// TIA Portal V16 export
// export: Created 2021-11-12T13:31:07.6036051Z, ExportSetting WithDefaults, DisplayName Totally Integrated Automation Portal, DisplayVersion V16 Update 3, DisplayName TIA Portal Version Control Interface, DisplayVersion V16 Update 2, DisplayName TIA Portal Openness, DisplayVersion V16 Update 3, DisplayName SINAMICS Startdrive Advanced, DisplayVersion V16 Update 5, DisplayName SINAMICS Startdrive G130, G150, S120, S150, SINAMICS MV, S210, DisplayVersion V16 Update 5, DisplayName SINAMICS Startdrive G110M, G120, G120C, G120D, G120P, G115D, DisplayVersion V16 Update 5, DisplayName STEP 7 Professional, DisplayVersion V16 Update 3, DisplayName STEP 7 Safety, DisplayVersion V16, DisplayName WinCC UA Professional, DisplayVersion V16 Update 3
FUNCTION_BLOCK "Sfty_IO_Module"   // FB68, F_LAD
{ S7_Optimized_Access := 'TRUE' }
VERSION : 0.1
// Safety module fault evaluation
// stored: AutoNumber true, IsIECCheckEnabled false, UDAEnableTagReadback false
   VAR
      SF_AckGlobal : ACK_GL;
   END_VAR
BEGIN

REGION Network 2: Acknowledgment for reintegration
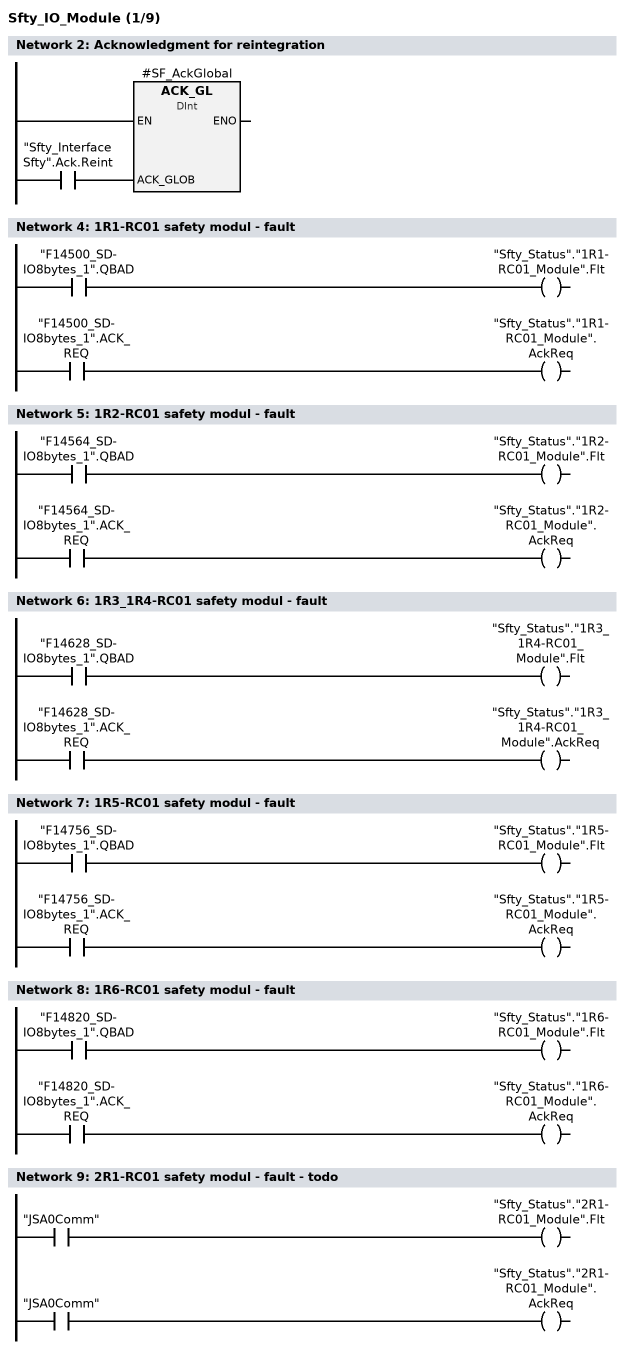
   RUNG wire#powerrail
      { S7_Templates := "codedbool_type := DInt" } #SF_AckGlobal.ACK_GL(ACK_GLOB := wire#w1)
   END_RUNG
   RUNG wire#powerrail
      Contact( "Sfty_InterfaceSfty".Ack.Reint )
   END_RUNG wire#w1
   // the same network as SCL:
   #SF_AckGlobal(ACK_GLOB := "Sfty_InterfaceSfty".Ack.Reint);   // ACK_GL
END_REGION

REGION Network 3: *************** Robot safety module fault ***************
END_REGION

REGION Network 4: 1R1-RC01 safety modul - fault
   RUNG wire#powerrail
      Contact( "F14500_SD-IO8bytes_1".QBAD )
      Coil( "Sfty_Status"."1R1-RC01_Module".Flt )
   END_RUNG
   RUNG wire#powerrail
      Contact( "F14500_SD-IO8bytes_1".ACK_REQ )
      Coil( "Sfty_Status"."1R1-RC01_Module".AckReq )
   END_RUNG
   // the same network as SCL:
   "Sfty_Status"."1R1-RC01_Module".Flt := "F14500_SD-IO8bytes_1".QBAD;
   "Sfty_Status"."1R1-RC01_Module".AckReq := "F14500_SD-IO8bytes_1".ACK_REQ;
END_REGION

REGION Network 5: 1R2-RC01 safety modul - fault
   RUNG wire#powerrail
      Contact( "F14564_SD-IO8bytes_1".QBAD )
      Coil( "Sfty_Status"."1R2-RC01_Module".Flt )
   END_RUNG
   RUNG wire#powerrail
      Contact( "F14564_SD-IO8bytes_1".ACK_REQ )
      Coil( "Sfty_Status"."1R2-RC01_Module".AckReq )
   END_RUNG
   // the same network as SCL:
   "Sfty_Status"."1R2-RC01_Module".Flt := "F14564_SD-IO8bytes_1".QBAD;
   "Sfty_Status"."1R2-RC01_Module".AckReq := "F14564_SD-IO8bytes_1".ACK_REQ;
END_REGION

REGION Network 6: 1R3_1R4-RC01 safety modul - fault
   RUNG wire#powerrail
      Contact( "F14628_SD-IO8bytes_1".QBAD )
      Coil( "Sfty_Status"."1R3_1R4-RC01_Module".Flt )
   END_RUNG
   RUNG wire#powerrail
      Contact( "F14628_SD-IO8bytes_1".ACK_REQ )
      Coil( "Sfty_Status"."1R3_1R4-RC01_Module".AckReq )
   END_RUNG
   // the same network as SCL:
   "Sfty_Status"."1R3_1R4-RC01_Module".Flt := "F14628_SD-IO8bytes_1".QBAD;
   "Sfty_Status"."1R3_1R4-RC01_Module".AckReq := "F14628_SD-IO8bytes_1".ACK_REQ;
END_REGION

REGION Network 7: 1R5-RC01 safety modul - fault
   RUNG wire#powerrail
      Contact( "F14756_SD-IO8bytes_1".QBAD )
      Coil( "Sfty_Status"."1R5-RC01_Module".Flt )
   END_RUNG
   RUNG wire#powerrail
      Contact( "F14756_SD-IO8bytes_1".ACK_REQ )
      Coil( "Sfty_Status"."1R5-RC01_Module".AckReq )
   END_RUNG
   // the same network as SCL:
   "Sfty_Status"."1R5-RC01_Module".Flt := "F14756_SD-IO8bytes_1".QBAD;
   "Sfty_Status"."1R5-RC01_Module".AckReq := "F14756_SD-IO8bytes_1".ACK_REQ;
END_REGION

REGION Network 8: 1R6-RC01 safety modul - fault
   RUNG wire#powerrail
      Contact( "F14820_SD-IO8bytes_1".QBAD )
      Coil( "Sfty_Status"."1R6-RC01_Module".Flt )
   END_RUNG
   RUNG wire#powerrail
      Contact( "F14820_SD-IO8bytes_1".ACK_REQ )
      Coil( "Sfty_Status"."1R6-RC01_Module".AckReq )
   END_RUNG
   // the same network as SCL:
   "Sfty_Status"."1R6-RC01_Module".Flt := "F14820_SD-IO8bytes_1".QBAD;
   "Sfty_Status"."1R6-RC01_Module".AckReq := "F14820_SD-IO8bytes_1".ACK_REQ;
END_REGION

REGION Network 9: 2R1-RC01 safety modul - fault - todo
   RUNG wire#powerrail
      Contact( "JSA0Comm" )
      Coil( "Sfty_Status"."2R1-RC01_Module".Flt )
   END_RUNG
   RUNG wire#powerrail
      Contact( "JSA0Comm" )
      Coil( "Sfty_Status"."2R1-RC01_Module".AckReq )
   END_RUNG
   // the same network as SCL:
   "Sfty_Status"."2R1-RC01_Module".Flt := "JSA0Comm";
   "Sfty_Status"."2R1-RC01_Module".AckReq := "JSA0Comm";
END_REGION

REGION Network 10: 2R2-RC01 safety modul - fault - todo
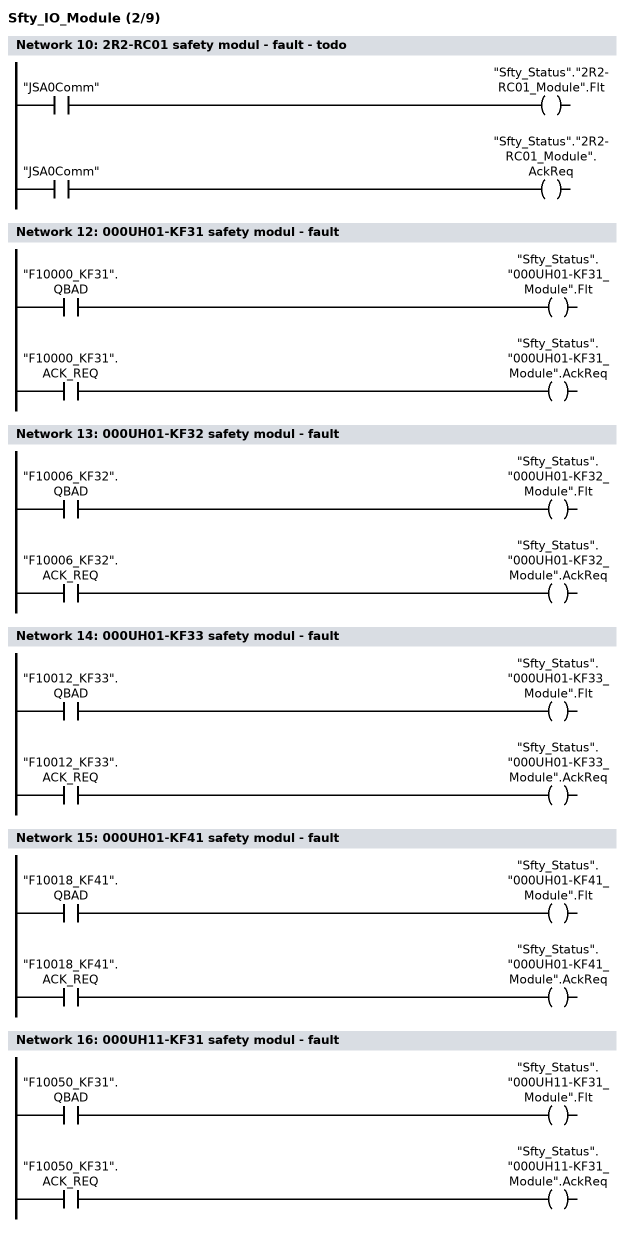
   RUNG wire#powerrail
      Contact( "JSA0Comm" )
      Coil( "Sfty_Status"."2R2-RC01_Module".Flt )
   END_RUNG
   RUNG wire#powerrail
      Contact( "JSA0Comm" )
      Coil( "Sfty_Status"."2R2-RC01_Module".AckReq )
   END_RUNG
   // the same network as SCL:
   "Sfty_Status"."2R2-RC01_Module".Flt := "JSA0Comm";
   "Sfty_Status"."2R2-RC01_Module".AckReq := "JSA0Comm";
END_REGION

REGION Network 11: *************** Input safety module fault ***************
END_REGION

REGION Network 12: 000UH01-KF31 safety modul - fault
   RUNG wire#powerrail
      Contact( "F10000_KF31".QBAD )
      Coil( "Sfty_Status"."000UH01-KF31_Module".Flt )
   END_RUNG
   RUNG wire#powerrail
      Contact( "F10000_KF31".ACK_REQ )
      Coil( "Sfty_Status"."000UH01-KF31_Module".AckReq )
   END_RUNG
   // the same network as SCL:
   "Sfty_Status"."000UH01-KF31_Module".Flt := "F10000_KF31".QBAD;
   "Sfty_Status"."000UH01-KF31_Module".AckReq := "F10000_KF31".ACK_REQ;
END_REGION

REGION Network 13: 000UH01-KF32 safety modul - fault
   RUNG wire#powerrail
      Contact( "F10006_KF32".QBAD )
      Coil( "Sfty_Status"."000UH01-KF32_Module".Flt )
   END_RUNG
   RUNG wire#powerrail
      Contact( "F10006_KF32".ACK_REQ )
      Coil( "Sfty_Status"."000UH01-KF32_Module".AckReq )
   END_RUNG
   // the same network as SCL:
   "Sfty_Status"."000UH01-KF32_Module".Flt := "F10006_KF32".QBAD;
   "Sfty_Status"."000UH01-KF32_Module".AckReq := "F10006_KF32".ACK_REQ;
END_REGION

REGION Network 14: 000UH01-KF33 safety modul - fault
   RUNG wire#powerrail
      Contact( "F10012_KF33".QBAD )
      Coil( "Sfty_Status"."000UH01-KF33_Module".Flt )
   END_RUNG
   RUNG wire#powerrail
      Contact( "F10012_KF33".ACK_REQ )
      Coil( "Sfty_Status"."000UH01-KF33_Module".AckReq )
   END_RUNG
   // the same network as SCL:
   "Sfty_Status"."000UH01-KF33_Module".Flt := "F10012_KF33".QBAD;
   "Sfty_Status"."000UH01-KF33_Module".AckReq := "F10012_KF33".ACK_REQ;
END_REGION

REGION Network 15: 000UH01-KF41 safety modul - fault
   RUNG wire#powerrail
      Contact( "F10018_KF41".QBAD )
      Coil( "Sfty_Status"."000UH01-KF41_Module".Flt )
   END_RUNG
   RUNG wire#powerrail
      Contact( "F10018_KF41".ACK_REQ )
      Coil( "Sfty_Status"."000UH01-KF41_Module".AckReq )
   END_RUNG
   // the same network as SCL:
   "Sfty_Status"."000UH01-KF41_Module".Flt := "F10018_KF41".QBAD;
   "Sfty_Status"."000UH01-KF41_Module".AckReq := "F10018_KF41".ACK_REQ;
END_REGION

REGION Network 16: 000UH11-KF31 safety modul - fault
   RUNG wire#powerrail
      Contact( "F10050_KF31".QBAD )
      Coil( "Sfty_Status"."000UH11-KF31_Module".Flt )
   END_RUNG
   RUNG wire#powerrail
      Contact( "F10050_KF31".ACK_REQ )
      Coil( "Sfty_Status"."000UH11-KF31_Module".AckReq )
   END_RUNG
   // the same network as SCL:
   "Sfty_Status"."000UH11-KF31_Module".Flt := "F10050_KF31".QBAD;
   "Sfty_Status"."000UH11-KF31_Module".AckReq := "F10050_KF31".ACK_REQ;
END_REGION

REGION Network 17: 000UH11-KF32 safety modul - fault
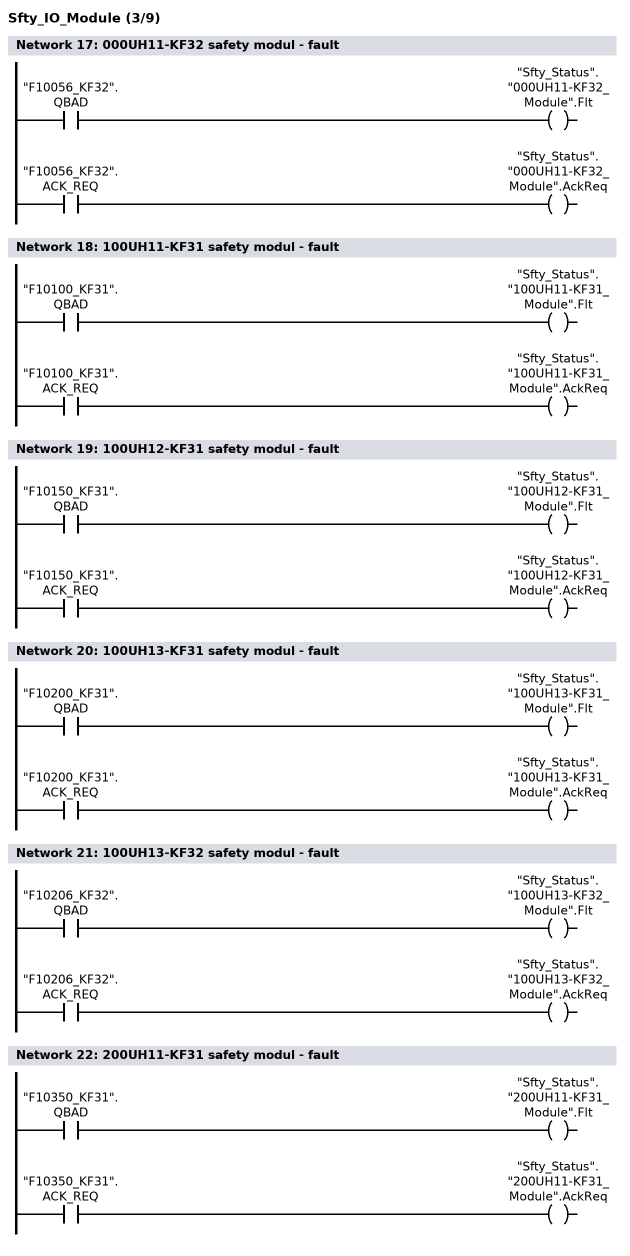
   RUNG wire#powerrail
      Contact( "F10056_KF32".QBAD )
      Coil( "Sfty_Status"."000UH11-KF32_Module".Flt )
   END_RUNG
   RUNG wire#powerrail
      Contact( "F10056_KF32".ACK_REQ )
      Coil( "Sfty_Status"."000UH11-KF32_Module".AckReq )
   END_RUNG
   // the same network as SCL:
   "Sfty_Status"."000UH11-KF32_Module".Flt := "F10056_KF32".QBAD;
   "Sfty_Status"."000UH11-KF32_Module".AckReq := "F10056_KF32".ACK_REQ;
END_REGION

REGION Network 18: 100UH11-KF31 safety modul - fault
   RUNG wire#powerrail
      Contact( "F10100_KF31".QBAD )
      Coil( "Sfty_Status"."100UH11-KF31_Module".Flt )
   END_RUNG
   RUNG wire#powerrail
      Contact( "F10100_KF31".ACK_REQ )
      Coil( "Sfty_Status"."100UH11-KF31_Module".AckReq )
   END_RUNG
   // the same network as SCL:
   "Sfty_Status"."100UH11-KF31_Module".Flt := "F10100_KF31".QBAD;
   "Sfty_Status"."100UH11-KF31_Module".AckReq := "F10100_KF31".ACK_REQ;
END_REGION

REGION Network 19: 100UH12-KF31 safety modul - fault
   RUNG wire#powerrail
      Contact( "F10150_KF31".QBAD )
      Coil( "Sfty_Status"."100UH12-KF31_Module".Flt )
   END_RUNG
   RUNG wire#powerrail
      Contact( "F10150_KF31".ACK_REQ )
      Coil( "Sfty_Status"."100UH12-KF31_Module".AckReq )
   END_RUNG
   // the same network as SCL:
   "Sfty_Status"."100UH12-KF31_Module".Flt := "F10150_KF31".QBAD;
   "Sfty_Status"."100UH12-KF31_Module".AckReq := "F10150_KF31".ACK_REQ;
END_REGION

REGION Network 20: 100UH13-KF31 safety modul - fault
   RUNG wire#powerrail
      Contact( "F10200_KF31".QBAD )
      Coil( "Sfty_Status"."100UH13-KF31_Module".Flt )
   END_RUNG
   RUNG wire#powerrail
      Contact( "F10200_KF31".ACK_REQ )
      Coil( "Sfty_Status"."100UH13-KF31_Module".AckReq )
   END_RUNG
   // the same network as SCL:
   "Sfty_Status"."100UH13-KF31_Module".Flt := "F10200_KF31".QBAD;
   "Sfty_Status"."100UH13-KF31_Module".AckReq := "F10200_KF31".ACK_REQ;
END_REGION

REGION Network 21: 100UH13-KF32 safety modul - fault
   RUNG wire#powerrail
      Contact( "F10206_KF32".QBAD )
      Coil( "Sfty_Status"."100UH13-KF32_Module".Flt )
   END_RUNG
   RUNG wire#powerrail
      Contact( "F10206_KF32".ACK_REQ )
      Coil( "Sfty_Status"."100UH13-KF32_Module".AckReq )
   END_RUNG
   // the same network as SCL:
   "Sfty_Status"."100UH13-KF32_Module".Flt := "F10206_KF32".QBAD;
   "Sfty_Status"."100UH13-KF32_Module".AckReq := "F10206_KF32".ACK_REQ;
END_REGION

REGION Network 22: 200UH11-KF31 safety modul - fault
   RUNG wire#powerrail
      Contact( "F10350_KF31".QBAD )
      Coil( "Sfty_Status"."200UH11-KF31_Module".Flt )
   END_RUNG
   RUNG wire#powerrail
      Contact( "F10350_KF31".ACK_REQ )
      Coil( "Sfty_Status"."200UH11-KF31_Module".AckReq )
   END_RUNG
   // the same network as SCL:
   "Sfty_Status"."200UH11-KF31_Module".Flt := "F10350_KF31".QBAD;
   "Sfty_Status"."200UH11-KF31_Module".AckReq := "F10350_KF31".ACK_REQ;
END_REGION

REGION Network 23: 300UH11-KF31 safety modul - fault
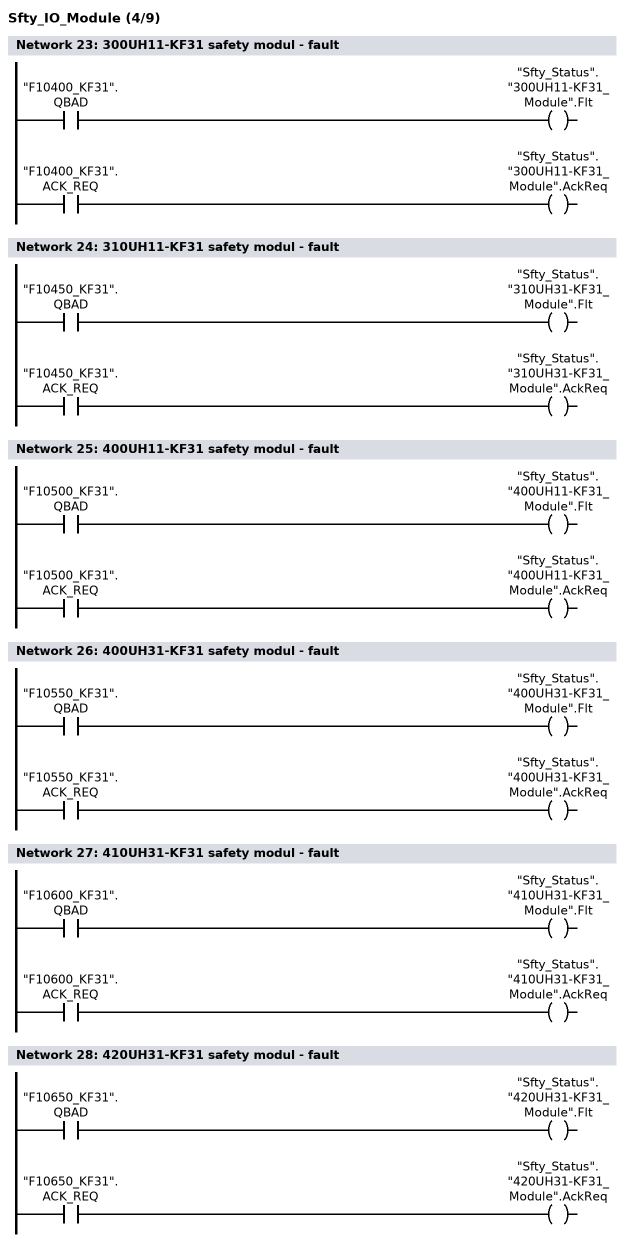
   RUNG wire#powerrail
      Contact( "F10400_KF31".QBAD )
      Coil( "Sfty_Status"."300UH11-KF31_Module".Flt )
   END_RUNG
   RUNG wire#powerrail
      Contact( "F10400_KF31".ACK_REQ )
      Coil( "Sfty_Status"."300UH11-KF31_Module".AckReq )
   END_RUNG
   // the same network as SCL:
   "Sfty_Status"."300UH11-KF31_Module".Flt := "F10400_KF31".QBAD;
   "Sfty_Status"."300UH11-KF31_Module".AckReq := "F10400_KF31".ACK_REQ;
END_REGION

REGION Network 24: 310UH11-KF31 safety modul - fault
   RUNG wire#powerrail
      Contact( "F10450_KF31".QBAD )
      Coil( "Sfty_Status"."310UH31-KF31_Module".Flt )
   END_RUNG
   RUNG wire#powerrail
      Contact( "F10450_KF31".ACK_REQ )
      Coil( "Sfty_Status"."310UH31-KF31_Module".AckReq )
   END_RUNG
   // the same network as SCL:
   "Sfty_Status"."310UH31-KF31_Module".Flt := "F10450_KF31".QBAD;
   "Sfty_Status"."310UH31-KF31_Module".AckReq := "F10450_KF31".ACK_REQ;
END_REGION

REGION Network 25: 400UH11-KF31 safety modul - fault
   RUNG wire#powerrail
      Contact( "F10500_KF31".QBAD )
      Coil( "Sfty_Status"."400UH11-KF31_Module".Flt )
   END_RUNG
   RUNG wire#powerrail
      Contact( "F10500_KF31".ACK_REQ )
      Coil( "Sfty_Status"."400UH11-KF31_Module".AckReq )
   END_RUNG
   // the same network as SCL:
   "Sfty_Status"."400UH11-KF31_Module".Flt := "F10500_KF31".QBAD;
   "Sfty_Status"."400UH11-KF31_Module".AckReq := "F10500_KF31".ACK_REQ;
END_REGION

REGION Network 26: 400UH31-KF31 safety modul - fault
   RUNG wire#powerrail
      Contact( "F10550_KF31".QBAD )
      Coil( "Sfty_Status"."400UH31-KF31_Module".Flt )
   END_RUNG
   RUNG wire#powerrail
      Contact( "F10550_KF31".ACK_REQ )
      Coil( "Sfty_Status"."400UH31-KF31_Module".AckReq )
   END_RUNG
   // the same network as SCL:
   "Sfty_Status"."400UH31-KF31_Module".Flt := "F10550_KF31".QBAD;
   "Sfty_Status"."400UH31-KF31_Module".AckReq := "F10550_KF31".ACK_REQ;
END_REGION

REGION Network 27: 410UH31-KF31 safety modul - fault
   RUNG wire#powerrail
      Contact( "F10600_KF31".QBAD )
      Coil( "Sfty_Status"."410UH31-KF31_Module".Flt )
   END_RUNG
   RUNG wire#powerrail
      Contact( "F10600_KF31".ACK_REQ )
      Coil( "Sfty_Status"."410UH31-KF31_Module".AckReq )
   END_RUNG
   // the same network as SCL:
   "Sfty_Status"."410UH31-KF31_Module".Flt := "F10600_KF31".QBAD;
   "Sfty_Status"."410UH31-KF31_Module".AckReq := "F10600_KF31".ACK_REQ;
END_REGION

REGION Network 28: 420UH31-KF31 safety modul - fault
   RUNG wire#powerrail
      Contact( "F10650_KF31".QBAD )
      Coil( "Sfty_Status"."420UH31-KF31_Module".Flt )
   END_RUNG
   RUNG wire#powerrail
      Contact( "F10650_KF31".ACK_REQ )
      Coil( "Sfty_Status"."420UH31-KF31_Module".AckReq )
   END_RUNG
   // the same network as SCL:
   "Sfty_Status"."420UH31-KF31_Module".Flt := "F10650_KF31".QBAD;
   "Sfty_Status"."420UH31-KF31_Module".AckReq := "F10650_KF31".ACK_REQ;
END_REGION

REGION Network 29: *************** Locks safety module fault ***************
END_REGION

REGION Network 30: 100+RU01-KF01 lock safety modul - fault
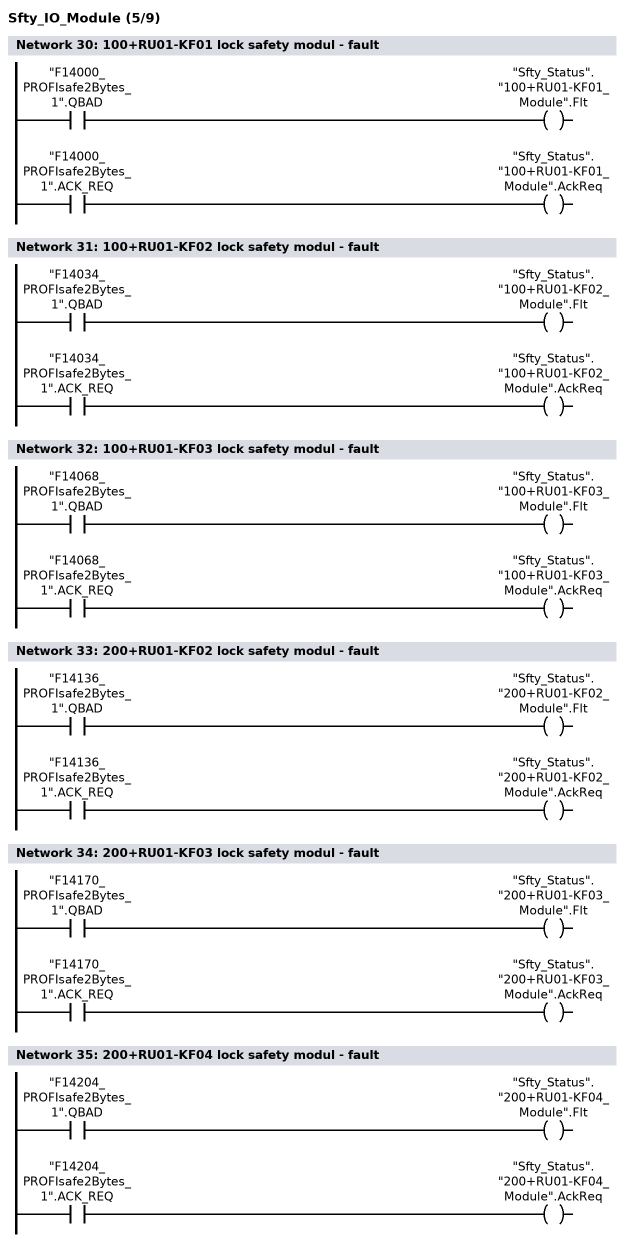
   RUNG wire#powerrail
      Contact( "F14000_PROFIsafe2Bytes_1".QBAD )
      Coil( "Sfty_Status"."100+RU01-KF01_Module".Flt )
   END_RUNG
   RUNG wire#powerrail
      Contact( "F14000_PROFIsafe2Bytes_1".ACK_REQ )
      Coil( "Sfty_Status"."100+RU01-KF01_Module".AckReq )
   END_RUNG
   // the same network as SCL:
   "Sfty_Status"."100+RU01-KF01_Module".Flt := "F14000_PROFIsafe2Bytes_1".QBAD;
   "Sfty_Status"."100+RU01-KF01_Module".AckReq := "F14000_PROFIsafe2Bytes_1".ACK_REQ;
END_REGION

REGION Network 31: 100+RU01-KF02 lock safety modul - fault
   RUNG wire#powerrail
      Contact( "F14034_PROFIsafe2Bytes_1".QBAD )
      Coil( "Sfty_Status"."100+RU01-KF02_Module".Flt )
   END_RUNG
   RUNG wire#powerrail
      Contact( "F14034_PROFIsafe2Bytes_1".ACK_REQ )
      Coil( "Sfty_Status"."100+RU01-KF02_Module".AckReq )
   END_RUNG
   // the same network as SCL:
   "Sfty_Status"."100+RU01-KF02_Module".Flt := "F14034_PROFIsafe2Bytes_1".QBAD;
   "Sfty_Status"."100+RU01-KF02_Module".AckReq := "F14034_PROFIsafe2Bytes_1".ACK_REQ;
END_REGION

REGION Network 32: 100+RU01-KF03 lock safety modul - fault
   RUNG wire#powerrail
      Contact( "F14068_PROFIsafe2Bytes_1".QBAD )
      Coil( "Sfty_Status"."100+RU01-KF03_Module".Flt )
   END_RUNG
   RUNG wire#powerrail
      Contact( "F14068_PROFIsafe2Bytes_1".ACK_REQ )
      Coil( "Sfty_Status"."100+RU01-KF03_Module".AckReq )
   END_RUNG
   // the same network as SCL:
   "Sfty_Status"."100+RU01-KF03_Module".Flt := "F14068_PROFIsafe2Bytes_1".QBAD;
   "Sfty_Status"."100+RU01-KF03_Module".AckReq := "F14068_PROFIsafe2Bytes_1".ACK_REQ;
END_REGION

REGION Network 33: 200+RU01-KF02 lock safety modul - fault
   RUNG wire#powerrail
      Contact( "F14136_PROFIsafe2Bytes_1".QBAD )
      Coil( "Sfty_Status"."200+RU01-KF02_Module".Flt )
   END_RUNG
   RUNG wire#powerrail
      Contact( "F14136_PROFIsafe2Bytes_1".ACK_REQ )
      Coil( "Sfty_Status"."200+RU01-KF02_Module".AckReq )
   END_RUNG
   // the same network as SCL:
   "Sfty_Status"."200+RU01-KF02_Module".Flt := "F14136_PROFIsafe2Bytes_1".QBAD;
   "Sfty_Status"."200+RU01-KF02_Module".AckReq := "F14136_PROFIsafe2Bytes_1".ACK_REQ;
END_REGION

REGION Network 34: 200+RU01-KF03 lock safety modul - fault
   RUNG wire#powerrail
      Contact( "F14170_PROFIsafe2Bytes_1".QBAD )
      Coil( "Sfty_Status"."200+RU01-KF03_Module".Flt )
   END_RUNG
   RUNG wire#powerrail
      Contact( "F14170_PROFIsafe2Bytes_1".ACK_REQ )
      Coil( "Sfty_Status"."200+RU01-KF03_Module".AckReq )
   END_RUNG
   // the same network as SCL:
   "Sfty_Status"."200+RU01-KF03_Module".Flt := "F14170_PROFIsafe2Bytes_1".QBAD;
   "Sfty_Status"."200+RU01-KF03_Module".AckReq := "F14170_PROFIsafe2Bytes_1".ACK_REQ;
END_REGION

REGION Network 35: 200+RU01-KF04 lock safety modul - fault
   RUNG wire#powerrail
      Contact( "F14204_PROFIsafe2Bytes_1".QBAD )
      Coil( "Sfty_Status"."200+RU01-KF04_Module".Flt )
   END_RUNG
   RUNG wire#powerrail
      Contact( "F14204_PROFIsafe2Bytes_1".ACK_REQ )
      Coil( "Sfty_Status"."200+RU01-KF04_Module".AckReq )
   END_RUNG
   // the same network as SCL:
   "Sfty_Status"."200+RU01-KF04_Module".Flt := "F14204_PROFIsafe2Bytes_1".QBAD;
   "Sfty_Status"."200+RU01-KF04_Module".AckReq := "F14204_PROFIsafe2Bytes_1".ACK_REQ;
END_REGION

REGION Network 36: *************** Inverters safety module fault ***************
END_REGION

REGION Network 37: Inverter safety module fault - 110+UC12-TA01
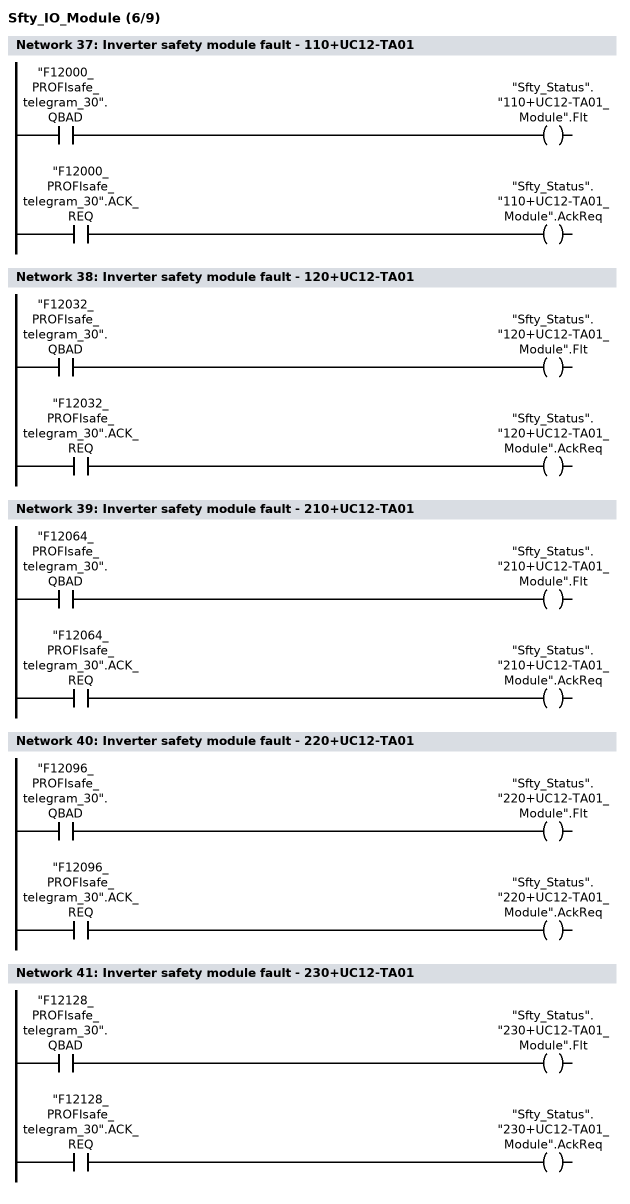
   RUNG wire#powerrail
      Contact( "F12000_PROFIsafe_telegram_30".QBAD )
      Coil( "Sfty_Status"."110+UC12-TA01_Module".Flt )
   END_RUNG
   RUNG wire#powerrail
      Contact( "F12000_PROFIsafe_telegram_30".ACK_REQ )
      Coil( "Sfty_Status"."110+UC12-TA01_Module".AckReq )
   END_RUNG
   // the same network as SCL:
   "Sfty_Status"."110+UC12-TA01_Module".Flt := "F12000_PROFIsafe_telegram_30".QBAD;
   "Sfty_Status"."110+UC12-TA01_Module".AckReq := "F12000_PROFIsafe_telegram_30".ACK_REQ;
END_REGION

REGION Network 38: Inverter safety module fault - 120+UC12-TA01
   RUNG wire#powerrail
      Contact( "F12032_PROFIsafe_telegram_30".QBAD )
      Coil( "Sfty_Status"."120+UC12-TA01_Module".Flt )
   END_RUNG
   RUNG wire#powerrail
      Contact( "F12032_PROFIsafe_telegram_30".ACK_REQ )
      Coil( "Sfty_Status"."120+UC12-TA01_Module".AckReq )
   END_RUNG
   // the same network as SCL:
   "Sfty_Status"."120+UC12-TA01_Module".Flt := "F12032_PROFIsafe_telegram_30".QBAD;
   "Sfty_Status"."120+UC12-TA01_Module".AckReq := "F12032_PROFIsafe_telegram_30".ACK_REQ;
END_REGION

REGION Network 39: Inverter safety module fault - 210+UC12-TA01
   RUNG wire#powerrail
      Contact( "F12064_PROFIsafe_telegram_30".QBAD )
      Coil( "Sfty_Status"."210+UC12-TA01_Module".Flt )
   END_RUNG
   RUNG wire#powerrail
      Contact( "F12064_PROFIsafe_telegram_30".ACK_REQ )
      Coil( "Sfty_Status"."210+UC12-TA01_Module".AckReq )
   END_RUNG
   // the same network as SCL:
   "Sfty_Status"."210+UC12-TA01_Module".Flt := "F12064_PROFIsafe_telegram_30".QBAD;
   "Sfty_Status"."210+UC12-TA01_Module".AckReq := "F12064_PROFIsafe_telegram_30".ACK_REQ;
END_REGION

REGION Network 40: Inverter safety module fault - 220+UC12-TA01
   RUNG wire#powerrail
      Contact( "F12096_PROFIsafe_telegram_30".QBAD )
      Coil( "Sfty_Status"."220+UC12-TA01_Module".Flt )
   END_RUNG
   RUNG wire#powerrail
      Contact( "F12096_PROFIsafe_telegram_30".ACK_REQ )
      Coil( "Sfty_Status"."220+UC12-TA01_Module".AckReq )
   END_RUNG
   // the same network as SCL:
   "Sfty_Status"."220+UC12-TA01_Module".Flt := "F12096_PROFIsafe_telegram_30".QBAD;
   "Sfty_Status"."220+UC12-TA01_Module".AckReq := "F12096_PROFIsafe_telegram_30".ACK_REQ;
END_REGION

REGION Network 41: Inverter safety module fault - 230+UC12-TA01
   RUNG wire#powerrail
      Contact( "F12128_PROFIsafe_telegram_30".QBAD )
      Coil( "Sfty_Status"."230+UC12-TA01_Module".Flt )
   END_RUNG
   RUNG wire#powerrail
      Contact( "F12128_PROFIsafe_telegram_30".ACK_REQ )
      Coil( "Sfty_Status"."230+UC12-TA01_Module".AckReq )
   END_RUNG
   // the same network as SCL:
   "Sfty_Status"."230+UC12-TA01_Module".Flt := "F12128_PROFIsafe_telegram_30".QBAD;
   "Sfty_Status"."230+UC12-TA01_Module".AckReq := "F12128_PROFIsafe_telegram_30".ACK_REQ;
END_REGION

REGION Network 42: Inverter safety module fault - 230+UC12-TA02
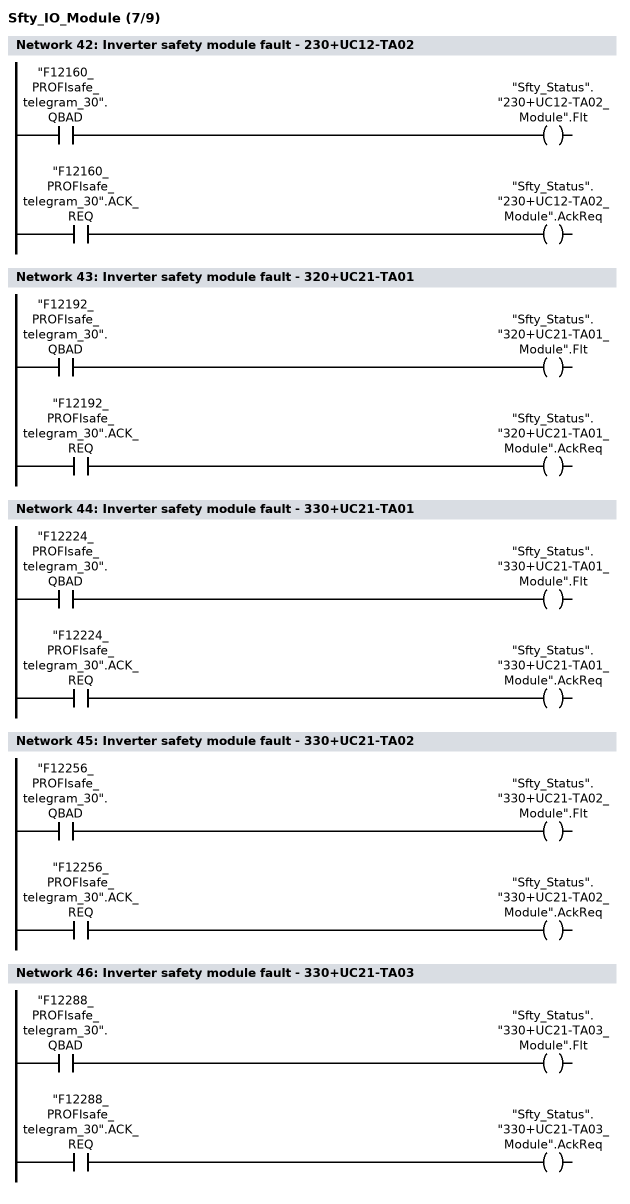
   RUNG wire#powerrail
      Contact( "F12160_PROFIsafe_telegram_30".QBAD )
      Coil( "Sfty_Status"."230+UC12-TA02_Module".Flt )
   END_RUNG
   RUNG wire#powerrail
      Contact( "F12160_PROFIsafe_telegram_30".ACK_REQ )
      Coil( "Sfty_Status"."230+UC12-TA02_Module".AckReq )
   END_RUNG
   // the same network as SCL:
   "Sfty_Status"."230+UC12-TA02_Module".Flt := "F12160_PROFIsafe_telegram_30".QBAD;
   "Sfty_Status"."230+UC12-TA02_Module".AckReq := "F12160_PROFIsafe_telegram_30".ACK_REQ;
END_REGION

REGION Network 43: Inverter safety module fault - 320+UC21-TA01
   RUNG wire#powerrail
      Contact( "F12192_PROFIsafe_telegram_30".QBAD )
      Coil( "Sfty_Status"."320+UC21-TA01_Module".Flt )
   END_RUNG
   RUNG wire#powerrail
      Contact( "F12192_PROFIsafe_telegram_30".ACK_REQ )
      Coil( "Sfty_Status"."320+UC21-TA01_Module".AckReq )
   END_RUNG
   // the same network as SCL:
   "Sfty_Status"."320+UC21-TA01_Module".Flt := "F12192_PROFIsafe_telegram_30".QBAD;
   "Sfty_Status"."320+UC21-TA01_Module".AckReq := "F12192_PROFIsafe_telegram_30".ACK_REQ;
END_REGION

REGION Network 44: Inverter safety module fault - 330+UC21-TA01
   RUNG wire#powerrail
      Contact( "F12224_PROFIsafe_telegram_30".QBAD )
      Coil( "Sfty_Status"."330+UC21-TA01_Module".Flt )
   END_RUNG
   RUNG wire#powerrail
      Contact( "F12224_PROFIsafe_telegram_30".ACK_REQ )
      Coil( "Sfty_Status"."330+UC21-TA01_Module".AckReq )
   END_RUNG
   // the same network as SCL:
   "Sfty_Status"."330+UC21-TA01_Module".Flt := "F12224_PROFIsafe_telegram_30".QBAD;
   "Sfty_Status"."330+UC21-TA01_Module".AckReq := "F12224_PROFIsafe_telegram_30".ACK_REQ;
END_REGION

REGION Network 45: Inverter safety module fault - 330+UC21-TA02
   RUNG wire#powerrail
      Contact( "F12256_PROFIsafe_telegram_30".QBAD )
      Coil( "Sfty_Status"."330+UC21-TA02_Module".Flt )
   END_RUNG
   RUNG wire#powerrail
      Contact( "F12256_PROFIsafe_telegram_30".ACK_REQ )
      Coil( "Sfty_Status"."330+UC21-TA02_Module".AckReq )
   END_RUNG
   // the same network as SCL:
   "Sfty_Status"."330+UC21-TA02_Module".Flt := "F12256_PROFIsafe_telegram_30".QBAD;
   "Sfty_Status"."330+UC21-TA02_Module".AckReq := "F12256_PROFIsafe_telegram_30".ACK_REQ;
END_REGION

REGION Network 46: Inverter safety module fault - 330+UC21-TA03
   RUNG wire#powerrail
      Contact( "F12288_PROFIsafe_telegram_30".QBAD )
      Coil( "Sfty_Status"."330+UC21-TA03_Module".Flt )
   END_RUNG
   RUNG wire#powerrail
      Contact( "F12288_PROFIsafe_telegram_30".ACK_REQ )
      Coil( "Sfty_Status"."330+UC21-TA03_Module".AckReq )
   END_RUNG
   // the same network as SCL:
   "Sfty_Status"."330+UC21-TA03_Module".Flt := "F12288_PROFIsafe_telegram_30".QBAD;
   "Sfty_Status"."330+UC21-TA03_Module".AckReq := "F12288_PROFIsafe_telegram_30".ACK_REQ;
END_REGION

REGION Network 47: Inverter safety module fault - 430+UC21-TA01
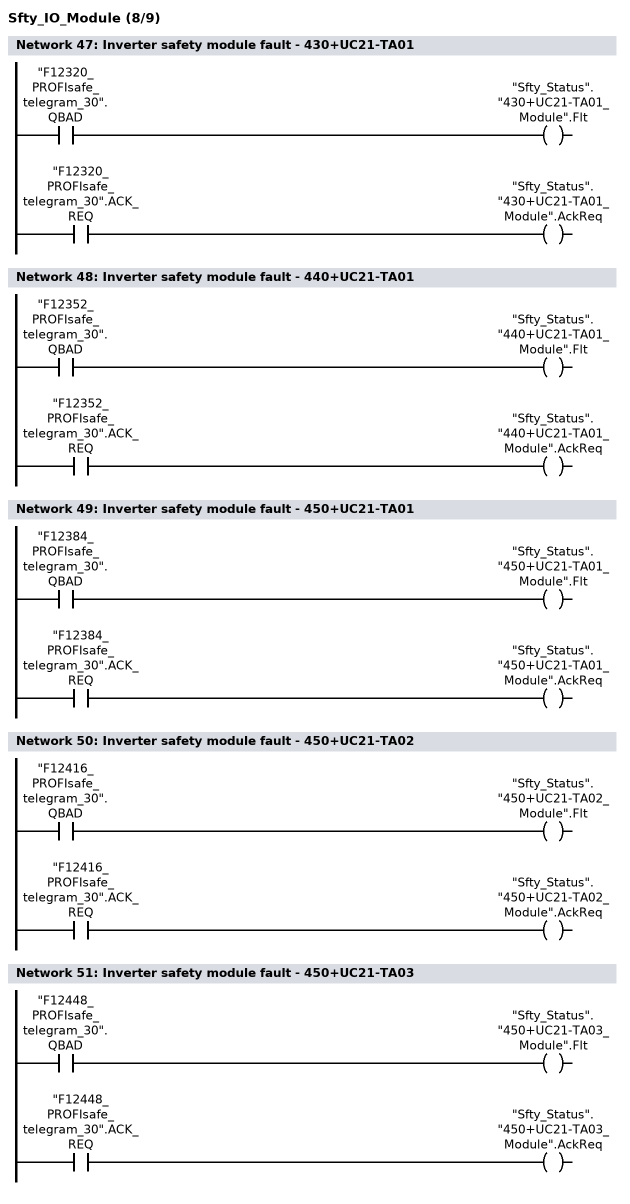
   RUNG wire#powerrail
      Contact( "F12320_PROFIsafe_telegram_30".QBAD )
      Coil( "Sfty_Status"."430+UC21-TA01_Module".Flt )
   END_RUNG
   RUNG wire#powerrail
      Contact( "F12320_PROFIsafe_telegram_30".ACK_REQ )
      Coil( "Sfty_Status"."430+UC21-TA01_Module".AckReq )
   END_RUNG
   // the same network as SCL:
   "Sfty_Status"."430+UC21-TA01_Module".Flt := "F12320_PROFIsafe_telegram_30".QBAD;
   "Sfty_Status"."430+UC21-TA01_Module".AckReq := "F12320_PROFIsafe_telegram_30".ACK_REQ;
END_REGION

REGION Network 48: Inverter safety module fault - 440+UC21-TA01
   RUNG wire#powerrail
      Contact( "F12352_PROFIsafe_telegram_30".QBAD )
      Coil( "Sfty_Status"."440+UC21-TA01_Module".Flt )
   END_RUNG
   RUNG wire#powerrail
      Contact( "F12352_PROFIsafe_telegram_30".ACK_REQ )
      Coil( "Sfty_Status"."440+UC21-TA01_Module".AckReq )
   END_RUNG
   // the same network as SCL:
   "Sfty_Status"."440+UC21-TA01_Module".Flt := "F12352_PROFIsafe_telegram_30".QBAD;
   "Sfty_Status"."440+UC21-TA01_Module".AckReq := "F12352_PROFIsafe_telegram_30".ACK_REQ;
END_REGION

REGION Network 49: Inverter safety module fault - 450+UC21-TA01
   RUNG wire#powerrail
      Contact( "F12384_PROFIsafe_telegram_30".QBAD )
      Coil( "Sfty_Status"."450+UC21-TA01_Module".Flt )
   END_RUNG
   RUNG wire#powerrail
      Contact( "F12384_PROFIsafe_telegram_30".ACK_REQ )
      Coil( "Sfty_Status"."450+UC21-TA01_Module".AckReq )
   END_RUNG
   // the same network as SCL:
   "Sfty_Status"."450+UC21-TA01_Module".Flt := "F12384_PROFIsafe_telegram_30".QBAD;
   "Sfty_Status"."450+UC21-TA01_Module".AckReq := "F12384_PROFIsafe_telegram_30".ACK_REQ;
END_REGION

REGION Network 50: Inverter safety module fault - 450+UC21-TA02
   RUNG wire#powerrail
      Contact( "F12416_PROFIsafe_telegram_30".QBAD )
      Coil( "Sfty_Status"."450+UC21-TA02_Module".Flt )
   END_RUNG
   RUNG wire#powerrail
      Contact( "F12416_PROFIsafe_telegram_30".ACK_REQ )
      Coil( "Sfty_Status"."450+UC21-TA02_Module".AckReq )
   END_RUNG
   // the same network as SCL:
   "Sfty_Status"."450+UC21-TA02_Module".Flt := "F12416_PROFIsafe_telegram_30".QBAD;
   "Sfty_Status"."450+UC21-TA02_Module".AckReq := "F12416_PROFIsafe_telegram_30".ACK_REQ;
END_REGION

REGION Network 51: Inverter safety module fault - 450+UC21-TA03
   RUNG wire#powerrail
      Contact( "F12448_PROFIsafe_telegram_30".QBAD )
      Coil( "Sfty_Status"."450+UC21-TA03_Module".Flt )
   END_RUNG
   RUNG wire#powerrail
      Contact( "F12448_PROFIsafe_telegram_30".ACK_REQ )
      Coil( "Sfty_Status"."450+UC21-TA03_Module".AckReq )
   END_RUNG
   // the same network as SCL:
   "Sfty_Status"."450+UC21-TA03_Module".Flt := "F12448_PROFIsafe_telegram_30".QBAD;
   "Sfty_Status"."450+UC21-TA03_Module".AckReq := "F12448_PROFIsafe_telegram_30".ACK_REQ;
END_REGION

REGION Network 52: Inverter safety module fault - 450+UC21-TA04
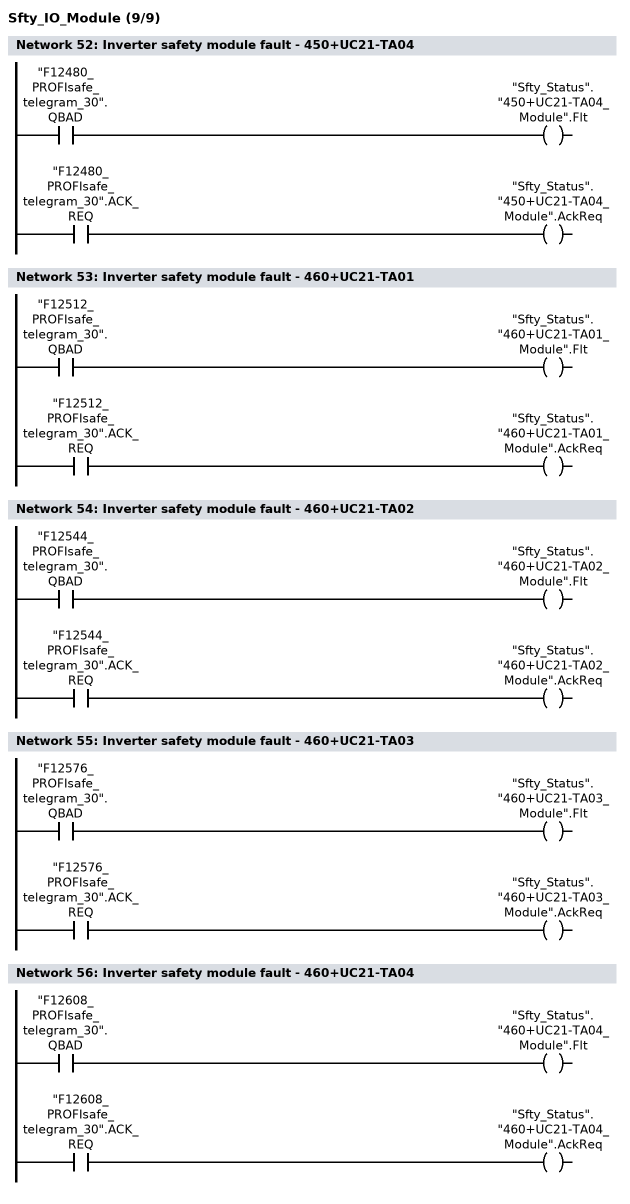
   RUNG wire#powerrail
      Contact( "F12480_PROFIsafe_telegram_30".QBAD )
      Coil( "Sfty_Status"."450+UC21-TA04_Module".Flt )
   END_RUNG
   RUNG wire#powerrail
      Contact( "F12480_PROFIsafe_telegram_30".ACK_REQ )
      Coil( "Sfty_Status"."450+UC21-TA04_Module".AckReq )
   END_RUNG
   // the same network as SCL:
   "Sfty_Status"."450+UC21-TA04_Module".Flt := "F12480_PROFIsafe_telegram_30".QBAD;
   "Sfty_Status"."450+UC21-TA04_Module".AckReq := "F12480_PROFIsafe_telegram_30".ACK_REQ;
END_REGION

REGION Network 53: Inverter safety module fault - 460+UC21-TA01
   RUNG wire#powerrail
      Contact( "F12512_PROFIsafe_telegram_30".QBAD )
      Coil( "Sfty_Status"."460+UC21-TA01_Module".Flt )
   END_RUNG
   RUNG wire#powerrail
      Contact( "F12512_PROFIsafe_telegram_30".ACK_REQ )
      Coil( "Sfty_Status"."460+UC21-TA01_Module".AckReq )
   END_RUNG
   // the same network as SCL:
   "Sfty_Status"."460+UC21-TA01_Module".Flt := "F12512_PROFIsafe_telegram_30".QBAD;
   "Sfty_Status"."460+UC21-TA01_Module".AckReq := "F12512_PROFIsafe_telegram_30".ACK_REQ;
END_REGION

REGION Network 54: Inverter safety module fault - 460+UC21-TA02
   RUNG wire#powerrail
      Contact( "F12544_PROFIsafe_telegram_30".QBAD )
      Coil( "Sfty_Status"."460+UC21-TA02_Module".Flt )
   END_RUNG
   RUNG wire#powerrail
      Contact( "F12544_PROFIsafe_telegram_30".ACK_REQ )
      Coil( "Sfty_Status"."460+UC21-TA02_Module".AckReq )
   END_RUNG
   // the same network as SCL:
   "Sfty_Status"."460+UC21-TA02_Module".Flt := "F12544_PROFIsafe_telegram_30".QBAD;
   "Sfty_Status"."460+UC21-TA02_Module".AckReq := "F12544_PROFIsafe_telegram_30".ACK_REQ;
END_REGION

REGION Network 55: Inverter safety module fault - 460+UC21-TA03
   RUNG wire#powerrail
      Contact( "F12576_PROFIsafe_telegram_30".QBAD )
      Coil( "Sfty_Status"."460+UC21-TA03_Module".Flt )
   END_RUNG
   RUNG wire#powerrail
      Contact( "F12576_PROFIsafe_telegram_30".ACK_REQ )
      Coil( "Sfty_Status"."460+UC21-TA03_Module".AckReq )
   END_RUNG
   // the same network as SCL:
   "Sfty_Status"."460+UC21-TA03_Module".Flt := "F12576_PROFIsafe_telegram_30".QBAD;
   "Sfty_Status"."460+UC21-TA03_Module".AckReq := "F12576_PROFIsafe_telegram_30".ACK_REQ;
END_REGION

REGION Network 56: Inverter safety module fault - 460+UC21-TA04
   RUNG wire#powerrail
      Contact( "F12608_PROFIsafe_telegram_30".QBAD )
      Coil( "Sfty_Status"."460+UC21-TA04_Module".Flt )
   END_RUNG
   RUNG wire#powerrail
      Contact( "F12608_PROFIsafe_telegram_30".ACK_REQ )
      Coil( "Sfty_Status"."460+UC21-TA04_Module".AckReq )
   END_RUNG
   // the same network as SCL:
   "Sfty_Status"."460+UC21-TA04_Module".Flt := "F12608_PROFIsafe_telegram_30".QBAD;
   "Sfty_Status"."460+UC21-TA04_Module".AckReq := "F12608_PROFIsafe_telegram_30".ACK_REQ;
END_REGION
END_FUNCTION_BLOCK
